(* CoDeSys 2.3 export: F_READ_SENSOR_TEMP.EXP *)

(* POU FUN/PARAMETERS/F_READ_SENSOR_TEMP, ST *)
FUNCTION F_READ_SENSOR_TEMP : BOOL
VAR_INPUT
END_VAR
VAR_IN_OUT
	stSensor : ST_SENSOR_TEMP;
	fbIdList : FB_IDLIST;
END_VAR
VAR
END_VAR
stSensor.Cal_K   := F_IDLIST_GETREAL( CONCAT(stSensor.Name, '_K'   ), fbIdList );
stSensor.Cal_Off := F_IDLIST_GETREAL( CONCAT(stSensor.Name, '_Off' ), fbIdList );

stSensor.LowDeg  := F_IDLIST_GETREAL( CONCAT(stSensor.Name, '_Mild' ), fbIdList );
stSensor.HigDeg  := F_IDLIST_GETREAL( CONCAT(stSensor.Name, '_High' ), fbIdList );
stSensor.MaxDeg  := F_IDLIST_GETREAL( CONCAT(stSensor.Name, '_Max'  ), fbIdList );
stSensor.Delay   := F_IDLIST_GETREAL( CONCAT(stSensor.Name, '_Dly'  ), fbIdList );
END_FUNCTION
